// TIA Portal V15.1 export
// export: Created 2024-05-17T05:38:40.3668408Z, ExportSetting WithDefaults, DisplayName Totally Integrated Automation Portal, DisplayVersion V15.1 Update 5, DisplayName TIA Portal Openness, DisplayVersion V15.1 Update 5, DisplayName SINAMICS Startdrive Advanced, DisplayVersion V15.1, DisplayName G130, G150, S120, S150, SINAMICS MV, S210, DisplayVersion V15.1, DisplayName G110M, G120, G120C, G120D, G120P, DisplayVersion V15.1, DisplayName STEP 7 Professional, DisplayVersion V15.1 Update 5, DisplayName STEP 7 Safety, DisplayVersion V15.1, DisplayName WinCC Professional, DisplayVersion V15.1 Update 5, DisplayName SIMATIC Visualization Architect, DisplayVersion V15.1
FUNCTION "LGBModelCode_Type2" : Void   // FC6602, FBD
TITLE = LModelCode_Type2
{ S7_Optimized_Access := 'TRUE' }
VERSION : 0.1
// ============================================================================
// This Module Splits The Model Code.
// ============================================================================
// stored: AutoNumber false, IsIECCheckEnabled false, SetENOAutomatically False, UDAEnableTagReadback false
   VAR_INPUT
      I_Enable : Bool;   // Enable Conversion
      I_MMFRUSS : DInt;   // Complete Modelcode
   END_VAR
   VAR_OUTPUT
      O_MM : Int;   // Part of the MMFRUSS (ModelCode)
      O_FR : Int;   // Part of the MMFRUSS (ModelCode)
      O_USS : Int;   // Part of the MMFRUSS (ModelCode)
      O_FRUSS : DInt;   // Part of the MMFRUSS (ModelCode)
      O_M1 : Int;   // Part of the MMFRUSS (ModelCode)
      O_M2 : Int;   // Part of the MMFRUSS (ModelCode)
      O_F : Int;   // Part of the MMFRUSS (ModelCode)
      O_R : Int;   // Part of the MMFRUSS (ModelCode)
      O_U : Int;   // Part of the MMFRUSS (ModelCode)
      O_S1 : Int;   // Part of the MMFRUSS (ModelCode)
      O_S2 : Int;   // Part of the MMFRUSS (ModelCode)
      O_Done : Bool;   // Splitting the model code has finished without error
      O_Error : Bool;   // Splitting the model code has finished with error
   END_VAR
   VAR_TEMP
      M1 : DInt;   // Part of the MMFRUSS (ModelCode)
      M2 : DInt;   // Part of the MMFRUSS (ModelCode)
      F : DInt;   // Part of the MMFRUSS (ModelCode)
      R : DInt;   // Part of the MMFRUSS (ModelCode)
      U : DInt;   // Part of the MMFRUSS (ModelCode)
      S1 : DInt;   // Part of the MMFRUSS (ModelCode)
      S2 : DInt;   // Part of the MMFRUSS (ModelCode)
      MMFRUSS : DInt;   // Intermediate result
      MFRUSS : DInt;   // Intermediate result
      FRUSS : DInt;   // Intermediate result
      RUSS : DInt;   // Intermediate result
      USS : DInt;   // Intermediate result
      MM : DInt;   // Intermediate result
      SS : DInt;   // Intermediate result
      FR : DInt;   // Intermediate result
      T_Int : Int;   // Intermediate result
      T_Dint : DInt;   // Intermediate result
   END_VAR
BEGIN

REGION Network 1: **** 4.2 - Machine Status - Parameter **** Reset temps
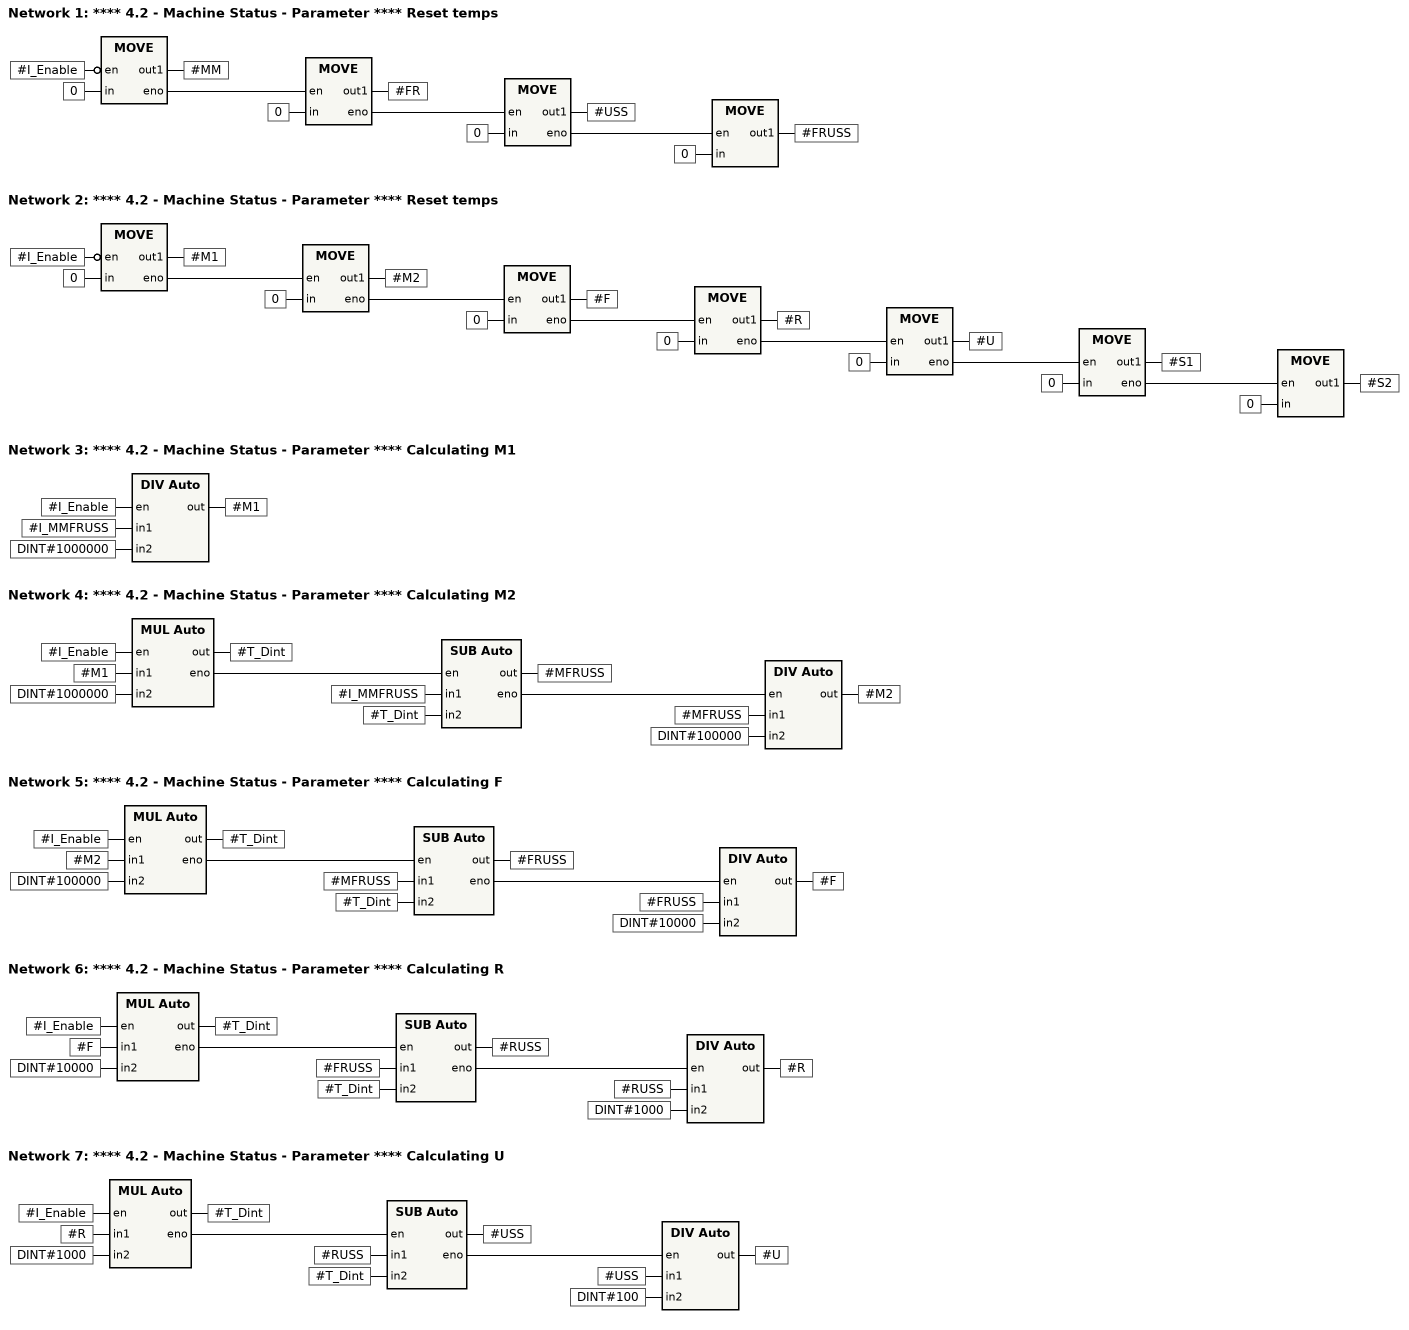
   IF NOT #I_Enable THEN
       #MM := 0;
       #FR := 0;
       #USS := 0;
       #FRUSS := 0;
   END_IF;
END_REGION

REGION Network 2: **** 4.2 - Machine Status - Parameter **** Reset temps
   IF NOT #I_Enable THEN
       #M1 := 0;
       #M2 := 0;
       #F := 0;
       #R := 0;
       #U := 0;
       #S1 := 0;
       #S2 := 0;
   END_IF;
END_REGION

REGION Network 3: **** 4.2 - Machine Status - Parameter **** Calculating M1
   IF #I_Enable THEN #M1 := #I_MMFRUSS / DINT#1000000; END_IF;
END_REGION

REGION Network 4: **** 4.2 - Machine Status - Parameter **** Calculating M2
   IF #I_Enable THEN
       #T_Dint := #M1 * DINT#1000000;
       #MFRUSS := #I_MMFRUSS - #T_Dint;
       #M2 := #MFRUSS / DINT#100000;
   END_IF;
END_REGION

REGION Network 5: **** 4.2 - Machine Status - Parameter **** Calculating F
   IF #I_Enable THEN
       #T_Dint := #M2 * DINT#100000;
       #FRUSS := #MFRUSS - #T_Dint;
       #F := #FRUSS / DINT#10000;
   END_IF;
END_REGION

REGION Network 6: **** 4.2 - Machine Status - Parameter **** Calculating R
   IF #I_Enable THEN
       #T_Dint := #F * DINT#10000;
       #RUSS := #FRUSS - #T_Dint;
       #R := #RUSS / DINT#1000;
   END_IF;
END_REGION

REGION Network 7: **** 4.2 - Machine Status - Parameter **** Calculating U
   IF #I_Enable THEN
       #T_Dint := #R * DINT#1000;
       #USS := #RUSS - #T_Dint;
       #U := #USS / DINT#100;
   END_IF;
END_REGION

REGION Network 8: **** 4.2 - Machine Status - Parameter **** Calculating S1
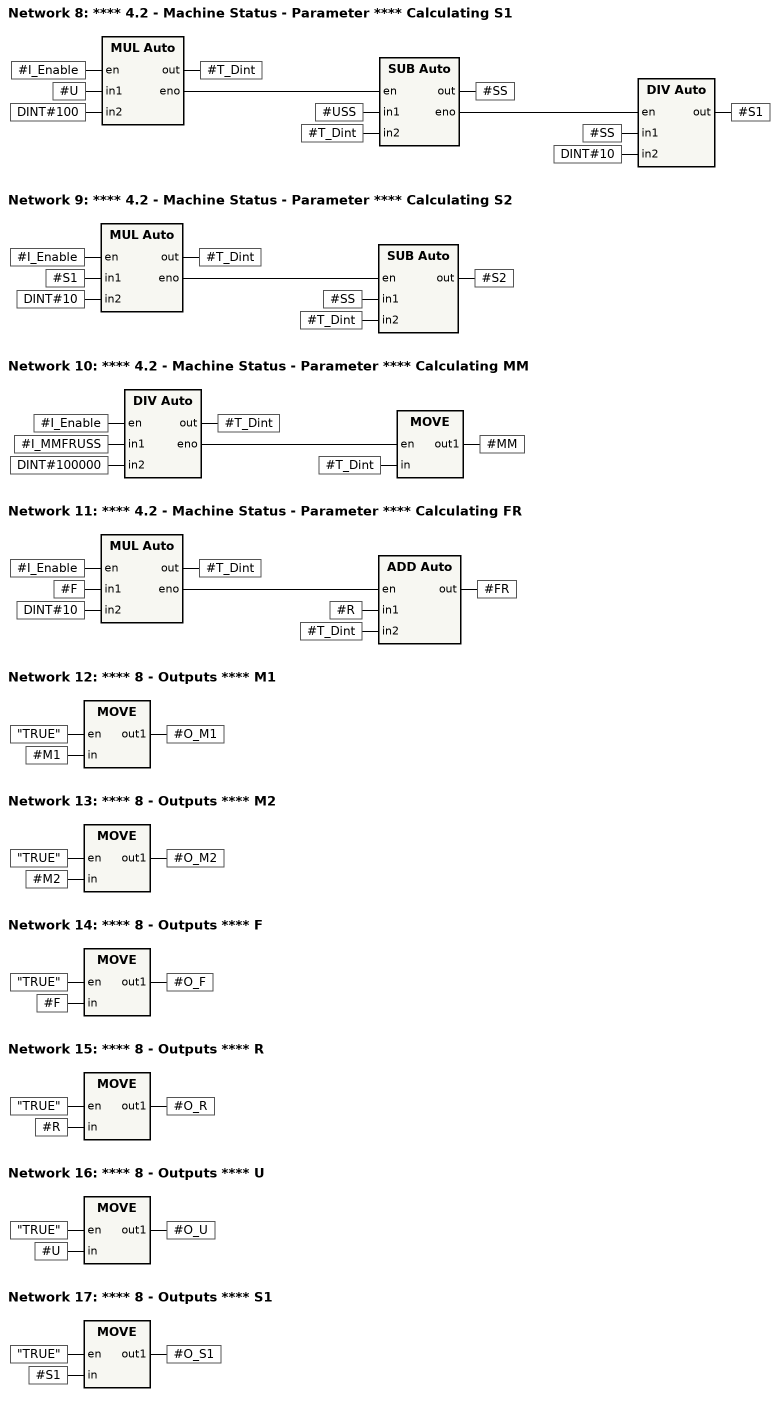
   IF #I_Enable THEN
       #T_Dint := #U * DINT#100;
       #SS := #USS - #T_Dint;
       #S1 := #SS / DINT#10;
   END_IF;
END_REGION

REGION Network 9: **** 4.2 - Machine Status - Parameter **** Calculating S2
   IF #I_Enable THEN
       #T_Dint := #S1 * DINT#10;
       #S2 := #SS - #T_Dint;
   END_IF;
END_REGION

REGION Network 10: **** 4.2 - Machine Status - Parameter **** Calculating MM
   IF #I_Enable THEN
       #T_Dint := #I_MMFRUSS / DINT#100000;
       #MM := #T_Dint;
   END_IF;
END_REGION

REGION Network 11: **** 4.2 - Machine Status - Parameter **** Calculating FR
   IF #I_Enable THEN
       #T_Dint := #F * DINT#10;
       #FR := #R + #T_Dint;
   END_IF;
END_REGION

REGION Network 12: **** 8 - Outputs **** M1
   IF "TRUE" THEN #O_M1 := #M1; END_IF;
END_REGION

REGION Network 13: **** 8 - Outputs **** M2
   IF "TRUE" THEN #O_M2 := #M2; END_IF;
END_REGION

REGION Network 14: **** 8 - Outputs **** F
   IF "TRUE" THEN #O_F := #F; END_IF;
END_REGION

REGION Network 15: **** 8 - Outputs **** R
   IF "TRUE" THEN #O_R := #R; END_IF;
END_REGION

REGION Network 16: **** 8 - Outputs **** U
   IF "TRUE" THEN #O_U := #U; END_IF;
END_REGION

REGION Network 17: **** 8 - Outputs **** S1
   IF "TRUE" THEN #O_S1 := #S1; END_IF;
END_REGION

REGION Network 18: **** 8 - Outputs **** S2
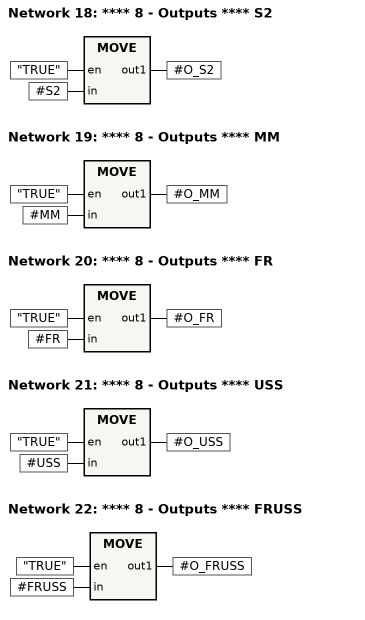
   IF "TRUE" THEN #O_S2 := #S2; END_IF;
END_REGION

REGION Network 19: **** 8 - Outputs **** MM
   IF "TRUE" THEN #O_MM := #MM; END_IF;
END_REGION

REGION Network 20: **** 8 - Outputs **** FR
   IF "TRUE" THEN #O_FR := #FR; END_IF;
END_REGION

REGION Network 21: **** 8 - Outputs **** USS
   IF "TRUE" THEN #O_USS := #USS; END_IF;
END_REGION

REGION Network 22: **** 8 - Outputs **** FRUSS
   IF "TRUE" THEN #O_FRUSS := #FRUSS; END_IF;
END_REGION
END_FUNCTION
